{attribute 'qualified_only'}
VAR_GLOBAL
	{attribute 'OPC.UA.DA' := '1'}
	{attribute 'OPC.UA.DA.StructuredType' := '1'}
	Alrm: DT_Incidences;

	
END_VAR

(* stored: Version 1.1.0.1, ProductVersion 3.1.4024.5
   GVL OPC_UA: Id {80a4bc94-1ad6-4926-890a-f214bb79f3d4} *)
